SUBAPPLICATION Uebung_080c (* Beispiel für E_CTU *)
  (* Standard: 61499-2; Description: Copyright (c) 2023 Meisterschulen am Ostbahnhof This program and the accompanying materials are made available under the terms of the Eclipse Public License 2.0 which is available at https://www.eclipse.org/legal/epl-2.0/ SPDX-License-Identifier: EPL-2.0 Beispiel für E_CTU Aufwärts zählen UAO Curriculum Module 3 - The IEC 61499 Standard, Seite 92 *)
  (* Version 1.0, 2023-10-23, Franz Höpfinger, Meisterschulen am Ostbahnhof *)
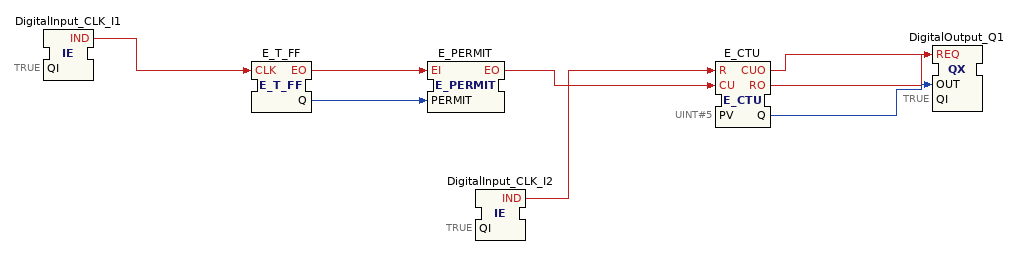
  (* Die Kombination von T_FF und PERMIT halbiert die Events. *)
  FBS
    DigitalOutput_Q1 : QX(QI := TRUE);
    DigitalInput_CLK_I1 : IE(QI := TRUE);
    E_CTU : E_CTU(PV := UINT#5);
    DigitalInput_CLK_I2 : IE(QI := TRUE);
    E_PERMIT : E_PERMIT;
    E_T_FF : E_T_FF;
  END_FBS
  EVENT_CONNECTIONS
    E_CTU.CUO TO DigitalOutput_Q1.REQ;
    E_CTU.RO TO DigitalOutput_Q1.REQ;
    DigitalInput_CLK_I2.IND TO E_CTU.R;
    E_T_FF.EO TO E_PERMIT.EI;
    DigitalInput_CLK_I1.IND TO E_T_FF.CLK;
    E_PERMIT.EO TO E_CTU.CU;
  END_CONNECTIONS
  DATA_CONNECTIONS
    E_CTU.Q TO DigitalOutput_Q1.OUT;
    E_T_FF.Q TO E_PERMIT.PERMIT;
  END_CONNECTIONS
END_SUBAPPLICATION
